FUNCTION_BLOCK GreenWhiteBackground (* Composite FB wrapping other FBs *)
  (* Standard: 61499-2 *)
  (* Version 1.0, 2022-11-10, franz *)
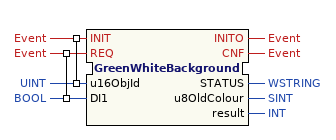
  EVENT_INPUT
    INIT WITH u16ObjId; (* Initialization Request *)
    REQ WITH DI1; (* Normal Execution Request *)
  END_EVENT
  EVENT_OUTPUT
    INITO; (* Initialization Confirm *)
    CNF; (* Execution Confirmation *)
  END_EVENT
  VAR_INPUT
    u16ObjId : UINT; (* Object ID *)
    DI1 : BOOL; (* Selelctor *)
  END_VAR
  VAR_OUTPUT
    STATUS : WSTRING; (* Service Status *)
    u8OldColour : SINT; (* Old value of ID *)
    result : INT; (* retval see description *)
  END_VAR
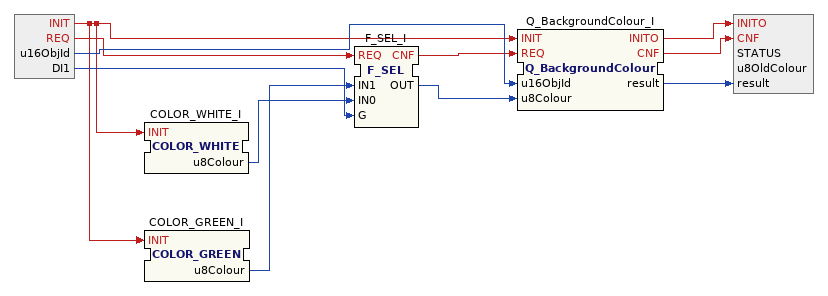
  FBS
    COLOR_GREEN_I : COLOR_GREEN;
    COLOR_WHITE_I : COLOR_WHITE;
    F_SEL_I : F_SEL;
    Q_BackgroundColour_I : Q_BackgroundColour;
  END_FBS
  EVENT_CONNECTIONS
    INIT TO COLOR_GREEN_I.INIT;
    INIT TO COLOR_WHITE_I.INIT;
    REQ TO F_SEL_I.REQ;
    INIT TO Q_BackgroundColour_I.INIT;
    F_SEL_I.CNF TO Q_BackgroundColour_I.REQ;
    Q_BackgroundColour_I.INITO TO INITO;
    Q_BackgroundColour_I.CNF TO CNF;
  END_CONNECTIONS
  DATA_CONNECTIONS
    COLOR_GREEN_I.u8Colour TO F_SEL_I.IN1;
    COLOR_WHITE_I.u8Colour TO F_SEL_I.IN0;
    DI1 TO F_SEL_I.G;
    u16ObjId TO Q_BackgroundColour_I.u16ObjId;
    F_SEL_I.OUT TO Q_BackgroundColour_I.u8Colour;
    Q_BackgroundColour_I.result TO result;
  END_CONNECTIONS
END_FUNCTION_BLOCK
